# EPICS substitutions: mpgSupport/Db/evgPatternIN20Test.substitutions
file bsaEdef.template {
  pattern { SYSI  , FBCK1 , FBCK2 , F1ID , F2ID , DEVICE       }
 	  { SYS0  , FBCK1 , FBCK2 , F1   , F2 ,  IOC:IN20:EV01 }
}
file evrPattern.template {
#	    Device        ,   Send SEQ RAM 1          PNET Processing LNK
  pattern { DEVICE        ,        LINK4             ,        LINK5         ,        LINK6           , LINKD }
	  { IOC:IN20:EV01 , "EVG:IN20:EV01:SEQ1SEND" , "IOC:IN20:EV01:PNET" , "IOC:IN20:EV01:EDEFFO" ,  ""   }
}
file bsaEVGmask.template {
  pattern { SYSI  ,  DEVICE       }
          { SYS0  , IOC:IN20:EV01 }
}
